DATA_BLOCK "DB_default_HMI"
{ DB_Accessible_From_Webserver := 'FALSE' ;
 S7_Optimized_Access := 'FALSE' }
VERSION : 0.1
NON_RETAIN
   STRUCT
      tALM { ExternalWritable := 'False'} : Struct   // HMI Alarms
         tE { ExternalWritable := 'False'} : Struct   // Stopping faults
            xSpare_0 { ExternalWritable := 'False'} : Bool;
            xSpare_1 { ExternalWritable := 'False'} : Bool;
            xSpare_2 { ExternalWritable := 'False'} : Bool;
            xSpare_3 { ExternalWritable := 'False'} : Bool;
            xSpare_4 { ExternalWritable := 'False'} : Bool;
            xSpare_5 { ExternalWritable := 'False'} : Bool;
            xSpare_6 { ExternalWritable := 'False'} : Bool;
            xSpare_7 { ExternalWritable := 'False'} : Bool;
            xSpare_8 { ExternalWritable := 'False'} : Bool;
            xSpare_9 { ExternalWritable := 'False'} : Bool;
            xSpare_10 { ExternalWritable := 'False'} : Bool;
            xSpare_11 { ExternalWritable := 'False'} : Bool;
            xSpare_12 { ExternalWritable := 'False'} : Bool;
            xSpare_13 { ExternalWritable := 'False'} : Bool;
            xSpare_14 { ExternalWritable := 'False'} : Bool;
            xSpare_15 { ExternalWritable := 'False'} : Bool;
            xSpare_16 { ExternalWritable := 'False'} : Bool;
            xSpare_17 { ExternalWritable := 'False'} : Bool;
            xSpare_18 { ExternalWritable := 'False'} : Bool;
            xSpare_19 { ExternalWritable := 'False'} : Bool;
            xSpare_20 { ExternalWritable := 'False'} : Bool;
            xSpare_21 { ExternalWritable := 'False'} : Bool;
            xSpare_22 { ExternalWritable := 'False'} : Bool;
            xSpare_23 { ExternalWritable := 'False'} : Bool;
            xSpare_24 { ExternalWritable := 'False'} : Bool;
            xSpare_25 { ExternalWritable := 'False'} : Bool;
            xSpare_26 { ExternalWritable := 'False'} : Bool;
            xSpare_27 { ExternalWritable := 'False'} : Bool;
            xSpare_28 { ExternalWritable := 'False'} : Bool;
            xSpare_29 { ExternalWritable := 'False'} : Bool;
            xSpare_30 { ExternalWritable := 'False'} : Bool;
            xSpare_31 { ExternalWritable := 'False'} : Bool;
         END_STRUCT;
         tS { ExternalWritable := 'False'} : Struct   // Stopping faults
            xLocalSafetySwitch { ExternalWritable := 'False'} : Bool;   // Local Safety Switch
            xFeedbackError { ExternalWritable := 'False'} : Bool;   // A171Az1.Feedback Error
            xDriveError { ExternalWritable := 'False'} : Bool;   // A171Az1.Drive Error
            xMotorFanProtection { ExternalWritable := 'False'} : Bool;   // A171QM1.Motor Fan protection
            xMotorThermalProbe { ExternalWritable := 'False'} : Bool;   // A547BT1.Motor Thermal Probe
            xSpare_5 { ExternalAccessible := 'False'; ExternalVisible := 'False'; ExternalWritable := 'False'} : Bool;
            xSpare_6 { ExternalAccessible := 'False'; ExternalVisible := 'False'; ExternalWritable := 'False'} : Bool;
            xSpare_7 { ExternalAccessible := 'False'; ExternalVisible := 'False'; ExternalWritable := 'False'} : Bool;
            xSpare_8 { ExternalAccessible := 'False'; ExternalVisible := 'False'; ExternalWritable := 'False'} : Bool;
            xSpare_9 { ExternalAccessible := 'False'; ExternalVisible := 'False'; ExternalWritable := 'False'} : Bool;
            xSpare_10 { ExternalAccessible := 'False'; ExternalVisible := 'False'; ExternalWritable := 'False'} : Bool;
            xSpare_11 { ExternalAccessible := 'False'; ExternalVisible := 'False'; ExternalWritable := 'False'} : Bool;
            xSpare_12 { ExternalAccessible := 'False'; ExternalVisible := 'False'; ExternalWritable := 'False'} : Bool;
            xSpare_13 { ExternalAccessible := 'False'; ExternalVisible := 'False'; ExternalWritable := 'False'} : Bool;
            xSpare_14 { ExternalAccessible := 'False'; ExternalVisible := 'False'; ExternalWritable := 'False'} : Bool;
            xSpare_15 { ExternalAccessible := 'False'; ExternalVisible := 'False'; ExternalWritable := 'False'} : Bool;
            xSpare_16 { ExternalAccessible := 'False'; ExternalVisible := 'False'; ExternalWritable := 'False'} : Bool;
            xSpare_17 { ExternalAccessible := 'False'; ExternalVisible := 'False'; ExternalWritable := 'False'} : Bool;
            xSpare_18 { ExternalAccessible := 'False'; ExternalVisible := 'False'; ExternalWritable := 'False'} : Bool;
            xSpare_19 { ExternalAccessible := 'False'; ExternalVisible := 'False'; ExternalWritable := 'False'} : Bool;
            xSpare_20 { ExternalAccessible := 'False'; ExternalVisible := 'False'; ExternalWritable := 'False'} : Bool;
            xSpare_21 { ExternalAccessible := 'False'; ExternalVisible := 'False'; ExternalWritable := 'False'} : Bool;
            xSpare_22 { ExternalAccessible := 'False'; ExternalVisible := 'False'; ExternalWritable := 'False'} : Bool;
            xSpare_23 { ExternalAccessible := 'False'; ExternalVisible := 'False'; ExternalWritable := 'False'} : Bool;
            xSpare_24 { ExternalAccessible := 'False'; ExternalVisible := 'False'; ExternalWritable := 'False'} : Bool;
            xSpare_25 { ExternalAccessible := 'False'; ExternalVisible := 'False'; ExternalWritable := 'False'} : Bool;
            xSpare_26 { ExternalAccessible := 'False'; ExternalVisible := 'False'; ExternalWritable := 'False'} : Bool;
            xSpare_27 { ExternalAccessible := 'False'; ExternalVisible := 'False'; ExternalWritable := 'False'} : Bool;
            xSpare_28 { ExternalAccessible := 'False'; ExternalVisible := 'False'; ExternalWritable := 'False'} : Bool;
            xSpare_29 { ExternalAccessible := 'False'; ExternalVisible := 'False'; ExternalWritable := 'False'} : Bool;
            xSpare_30 { ExternalAccessible := 'False'; ExternalVisible := 'False'; ExternalWritable := 'False'} : Bool;
            xSpare_31 { ExternalAccessible := 'False'; ExternalVisible := 'False'; ExternalWritable := 'False'} : Bool;
         END_STRUCT;
         tF { ExternalAccessible := 'False'; ExternalVisible := 'False'; ExternalWritable := 'False'} : Struct   // Faults
            xSpare_0 { ExternalAccessible := 'False'; ExternalVisible := 'False'; ExternalWritable := 'False'} : Bool;
            xSpare_1 { ExternalAccessible := 'False'; ExternalVisible := 'False'; ExternalWritable := 'False'} : Bool;
            xSpare_2 { ExternalAccessible := 'False'; ExternalVisible := 'False'; ExternalWritable := 'False'} : Bool;
            xSpare_3 { ExternalAccessible := 'False'; ExternalVisible := 'False'; ExternalWritable := 'False'} : Bool;
            xSpare_4 { ExternalAccessible := 'False'; ExternalVisible := 'False'; ExternalWritable := 'False'} : Bool;
            xSpare_5 { ExternalAccessible := 'False'; ExternalVisible := 'False'; ExternalWritable := 'False'} : Bool;
            xSpare_6 { ExternalAccessible := 'False'; ExternalVisible := 'False'; ExternalWritable := 'False'} : Bool;
            xSpare_7 { ExternalAccessible := 'False'; ExternalVisible := 'False'; ExternalWritable := 'False'} : Bool;
            xSpare_8 { ExternalAccessible := 'False'; ExternalVisible := 'False'; ExternalWritable := 'False'} : Bool;
            xSpare_9 { ExternalAccessible := 'False'; ExternalVisible := 'False'; ExternalWritable := 'False'} : Bool;
            xSpare_10 { ExternalAccessible := 'False'; ExternalVisible := 'False'; ExternalWritable := 'False'} : Bool;
            xSpare_11 { ExternalAccessible := 'False'; ExternalVisible := 'False'; ExternalWritable := 'False'} : Bool;
            xSpare_12 { ExternalAccessible := 'False'; ExternalVisible := 'False'; ExternalWritable := 'False'} : Bool;
            xSpare_13 { ExternalAccessible := 'False'; ExternalVisible := 'False'; ExternalWritable := 'False'} : Bool;
            xSpare_14 { ExternalAccessible := 'False'; ExternalVisible := 'False'; ExternalWritable := 'False'} : Bool;
            xSpare_15 { ExternalAccessible := 'False'; ExternalVisible := 'False'; ExternalWritable := 'False'} : Bool;
            xSpare_16 { ExternalAccessible := 'False'; ExternalVisible := 'False'; ExternalWritable := 'False'} : Bool;
            xSpare_17 { ExternalAccessible := 'False'; ExternalVisible := 'False'; ExternalWritable := 'False'} : Bool;
            xSpare_18 { ExternalAccessible := 'False'; ExternalVisible := 'False'; ExternalWritable := 'False'} : Bool;
            xSpare_19 { ExternalAccessible := 'False'; ExternalVisible := 'False'; ExternalWritable := 'False'} : Bool;
            xSpare_20 { ExternalAccessible := 'False'; ExternalVisible := 'False'; ExternalWritable := 'False'} : Bool;
            xSpare_21 { ExternalAccessible := 'False'; ExternalVisible := 'False'; ExternalWritable := 'False'} : Bool;
            xSpare_22 { ExternalAccessible := 'False'; ExternalVisible := 'False'; ExternalWritable := 'False'} : Bool;
            xSpare_23 { ExternalAccessible := 'False'; ExternalVisible := 'False'; ExternalWritable := 'False'} : Bool;
            xSpare_24 { ExternalAccessible := 'False'; ExternalVisible := 'False'; ExternalWritable := 'False'} : Bool;
            xSpare_25 { ExternalAccessible := 'False'; ExternalVisible := 'False'; ExternalWritable := 'False'} : Bool;
            xSpare_26 { ExternalAccessible := 'False'; ExternalVisible := 'False'; ExternalWritable := 'False'} : Bool;
            xSpare_27 { ExternalAccessible := 'False'; ExternalVisible := 'False'; ExternalWritable := 'False'} : Bool;
            xSpare_28 { ExternalAccessible := 'False'; ExternalVisible := 'False'; ExternalWritable := 'False'} : Bool;
            xSpare_29 { ExternalAccessible := 'False'; ExternalVisible := 'False'; ExternalWritable := 'False'} : Bool;
            xSpare_30 { ExternalAccessible := 'False'; ExternalVisible := 'False'; ExternalWritable := 'False'} : Bool;
            xSpare_31 { ExternalAccessible := 'False'; ExternalVisible := 'False'; ExternalWritable := 'False'} : Bool;
         END_STRUCT;
         tW { ExternalAccessible := 'False'; ExternalVisible := 'False'; ExternalWritable := 'False'} : Struct   // Warnings
            xSpare_0 { ExternalAccessible := 'False'; ExternalVisible := 'False'; ExternalWritable := 'False'} : Bool;
            xSpare_1 { ExternalAccessible := 'False'; ExternalVisible := 'False'; ExternalWritable := 'False'} : Bool;
            xSpare_2 { ExternalAccessible := 'False'; ExternalVisible := 'False'; ExternalWritable := 'False'} : Bool;
            xSpare_3 { ExternalAccessible := 'False'; ExternalVisible := 'False'; ExternalWritable := 'False'} : Bool;
            xSpare_4 { ExternalAccessible := 'False'; ExternalVisible := 'False'; ExternalWritable := 'False'} : Bool;
            xSpare_5 { ExternalAccessible := 'False'; ExternalVisible := 'False'; ExternalWritable := 'False'} : Bool;
            xSpare_6 { ExternalAccessible := 'False'; ExternalVisible := 'False'; ExternalWritable := 'False'} : Bool;
            xSpare_7 { ExternalAccessible := 'False'; ExternalVisible := 'False'; ExternalWritable := 'False'} : Bool;
            xSpare_8 { ExternalAccessible := 'False'; ExternalVisible := 'False'; ExternalWritable := 'False'} : Bool;
            xSpare_9 { ExternalAccessible := 'False'; ExternalVisible := 'False'; ExternalWritable := 'False'} : Bool;
            xSpare_10 { ExternalAccessible := 'False'; ExternalVisible := 'False'; ExternalWritable := 'False'} : Bool;
            xSpare_11 { ExternalAccessible := 'False'; ExternalVisible := 'False'; ExternalWritable := 'False'} : Bool;
            xSpare_12 { ExternalAccessible := 'False'; ExternalVisible := 'False'; ExternalWritable := 'False'} : Bool;
            xSpare_13 { ExternalAccessible := 'False'; ExternalVisible := 'False'; ExternalWritable := 'False'} : Bool;
            xSpare_14 { ExternalAccessible := 'False'; ExternalVisible := 'False'; ExternalWritable := 'False'} : Bool;
            xSpare_15 { ExternalAccessible := 'False'; ExternalVisible := 'False'; ExternalWritable := 'False'} : Bool;
            xSpare_16 { ExternalAccessible := 'False'; ExternalVisible := 'False'; ExternalWritable := 'False'} : Bool;
            xSpare_17 { ExternalAccessible := 'False'; ExternalVisible := 'False'; ExternalWritable := 'False'} : Bool;
            xSpare_18 { ExternalAccessible := 'False'; ExternalVisible := 'False'; ExternalWritable := 'False'} : Bool;
            xSpare_19 { ExternalAccessible := 'False'; ExternalVisible := 'False'; ExternalWritable := 'False'} : Bool;
            xSpare_20 { ExternalAccessible := 'False'; ExternalVisible := 'False'; ExternalWritable := 'False'} : Bool;
            xSpare_21 { ExternalAccessible := 'False'; ExternalVisible := 'False'; ExternalWritable := 'False'} : Bool;
            xSpare_22 { ExternalAccessible := 'False'; ExternalVisible := 'False'; ExternalWritable := 'False'} : Bool;
            xSpare_23 { ExternalAccessible := 'False'; ExternalVisible := 'False'; ExternalWritable := 'False'} : Bool;
            xSpare_24 { ExternalAccessible := 'False'; ExternalVisible := 'False'; ExternalWritable := 'False'} : Bool;
            xSpare_25 { ExternalAccessible := 'False'; ExternalVisible := 'False'; ExternalWritable := 'False'} : Bool;
            xSpare_26 { ExternalAccessible := 'False'; ExternalVisible := 'False'; ExternalWritable := 'False'} : Bool;
            xSpare_27 { ExternalAccessible := 'False'; ExternalVisible := 'False'; ExternalWritable := 'False'} : Bool;
            xSpare_28 { ExternalAccessible := 'False'; ExternalVisible := 'False'; ExternalWritable := 'False'} : Bool;
            xSpare_29 { ExternalAccessible := 'False'; ExternalVisible := 'False'; ExternalWritable := 'False'} : Bool;
            xSpare_30 { ExternalAccessible := 'False'; ExternalVisible := 'False'; ExternalWritable := 'False'} : Bool;
            xSpare_31 { ExternalAccessible := 'False'; ExternalVisible := 'False'; ExternalWritable := 'False'} : Bool;
         END_STRUCT;
      END_STRUCT;
      tHMR { ExternalWritable := 'False'} : Struct   // HMI Read
         xSpare0 { ExternalWritable := 'False'} : Bool;
         xSpare1 { ExternalWritable := 'False'} : Bool;
         xSpare2 { ExternalWritable := 'False'} : Bool;
         xSpare3 { ExternalWritable := 'False'} : Bool;
         xSpare4 { ExternalWritable := 'False'} : Bool;
         xSpare5 { ExternalWritable := 'False'} : Bool;
         xSpare6 { ExternalWritable := 'False'} : Bool;
         xSpare7 { ExternalWritable := 'False'} : Bool;
         xSpare8 { ExternalWritable := 'False'} : Bool;
         xSpare9 { ExternalWritable := 'False'} : Bool;
         xSpare10 { ExternalWritable := 'False'} : Bool;
         xSpare11 { ExternalWritable := 'False'} : Bool;
         xSpare12 { ExternalWritable := 'False'} : Bool;
         xSpare13 { ExternalWritable := 'False'} : Bool;
         xManualCommandEnabled { ExternalWritable := 'False'} : Bool;   // Manual Command enabled {x|x|x|x|O}
         xSpare15 { ExternalWritable := 'False'} : Bool;
         xSpare16 { ExternalWritable := 'False'} : Bool;
         xSpare17 { ExternalWritable := 'False'} : Bool;
         xSpare18 { ExternalWritable := 'False'} : Bool;
         xSpare19 { ExternalWritable := 'False'} : Bool;
         xSpare20 { ExternalWritable := 'False'} : Bool;
         xSpare21 { ExternalWritable := 'False'} : Bool;
         xSpare22 { ExternalWritable := 'False'} : Bool;
         xSpare23 { ExternalWritable := 'False'} : Bool;
         xSpare24 { ExternalWritable := 'False'} : Bool;
         xSpare25 { ExternalWritable := 'False'} : Bool;
         xSpare26 { ExternalWritable := 'False'} : Bool;
         xSpare27 { ExternalWritable := 'False'} : Bool;
         xSpare28 { ExternalWritable := 'False'} : Bool;
         xSpare29 { ExternalWritable := 'False'} : Bool;
         xSpare30 { ExternalWritable := 'False'} : Bool;
         xSpare31 { ExternalWritable := 'False'} : Bool;
         xSpare { ExternalWritable := 'False'} : Array[0..15] of Bool;
         iSpare0 { ExternalWritable := 'False'} : Int;
         iSpare1 { ExternalWritable := 'False'} : Int;
         iSpare2 { ExternalWritable := 'False'} : Int;
         iSpare3 { ExternalWritable := 'False'} : Int;
         iSpare4 { ExternalWritable := 'False'} : Int;
         iSpare5 { ExternalWritable := 'False'} : Int;
         iSpare6 { ExternalWritable := 'False'} : Int;
         iSpare7 { ExternalWritable := 'False'} : Int;
         iSpare8 { ExternalWritable := 'False'} : Int;
         iSpare9 { ExternalWritable := 'False'} : Int;
         iSpare10 { ExternalWritable := 'False'} : Int;
         iSpare11 { ExternalWritable := 'False'} : Int;
         iSpare12 { ExternalWritable := 'False'} : Int;
         iSpare13 { ExternalWritable := 'False'} : Int;
         iSpare14 { ExternalWritable := 'False'} : Int;
         iSpare15 { ExternalWritable := 'False'} : Int;
         iSpare16 { ExternalWritable := 'False'} : Int;
         dSpare0 { ExternalWritable := 'False'} : DInt;   //
         dSpare1 { ExternalWritable := 'False'} : DInt;   //
         dSpare2 { ExternalWritable := 'False'} : DInt;
         dSpare3 { ExternalWritable := 'False'} : DInt;
         dSpare4 { ExternalWritable := 'False'} : DInt;
         dSpare5 { ExternalWritable := 'False'} : DInt;
         dSpare6 { ExternalWritable := 'False'} : DInt;
         dSpare7 { ExternalWritable := 'False'} : DInt;
         dSpare8 { ExternalWritable := 'False'} : DInt;
         dSpare9 { ExternalWritable := 'False'} : DInt;
         dSpare10 { ExternalWritable := 'False'} : DInt;
         dSpare11 { ExternalWritable := 'False'} : DInt;
         dSpare12 { ExternalWritable := 'False'} : DInt;
         dSpare13 { ExternalWritable := 'False'} : DInt;
         dSpare14 { ExternalWritable := 'False'} : DInt;
         dSpare15 { ExternalWritable := 'False'} : DInt;
         rSpare0 { ExternalWritable := 'False'} : Real;
         rSpare1 { ExternalWritable := 'False'} : Real;
         rSpare2 { ExternalWritable := 'False'} : Real;
         rSpare3 { ExternalWritable := 'False'} : Real;
         rSpare4 { ExternalWritable := 'False'} : Real;
         rSpare5 { ExternalWritable := 'False'} : Real;
         rSpare6 { ExternalWritable := 'False'} : Real;
         rSpare7 { ExternalWritable := 'False'} : Real;
         rSpare8 { ExternalWritable := 'False'} : Real;
         tManCmd { ExternalWritable := 'False'} : Struct
            xSpare0 { ExternalWritable := 'False'} : Bool;   //
            xSpare1 { ExternalWritable := 'False'} : Bool;
            xSpare2 { ExternalWritable := 'False'} : Bool;
            xSpare3 { ExternalWritable := 'False'} : Bool;
            xSpare4 { ExternalWritable := 'False'} : Bool;
            xSpare5 { ExternalWritable := 'False'} : Bool;
            xSpare6 { ExternalWritable := 'False'} : Bool;
            xSpare7 { ExternalWritable := 'False'} : Bool;
            xSpare8 { ExternalWritable := 'False'} : Bool;
            xSpare9 { ExternalWritable := 'False'} : Bool;
            xSpare10 { ExternalWritable := 'False'} : Bool;
            xSpare11 { ExternalWritable := 'False'} : Bool;
            xSpare12 { ExternalWritable := 'False'} : Bool;
            xSpare13 { ExternalWritable := 'False'} : Bool;
            xSpare14 { ExternalWritable := 'False'} : Bool;
            xSpare15 { ExternalWritable := 'False'} : Bool;
            xSpare { ExternalWritable := 'False'} : Array[0..15] of Bool;
         END_STRUCT;
      END_STRUCT;
      tHMW : Struct   // HMI Write
         xSpare0 : Bool;   //
         xSpare1 : Bool;
         xSpare2 : Bool;
         xSpare3 : Bool;
         xSpare4 : Bool;
         xSpare5 : Bool;
         xSpare6 : Bool;
         xSpare7 : Bool;
         xSpare8 : Bool;
         xSpare9 : Bool;
         xSpare10 : Bool;   //
         xSpare11 : Bool;
         xSpare12 : Bool;
         xSpare13 : Bool;
         xEnableManualCommand : Bool;   // Enable Disable Manual command {x|x|x|x|O}
         xSpare15 : Bool;
         xSpare16 : Bool;
         xSpare17 : Bool;
         xSpare18 : Bool;
         xSpare19 : Bool;
         xSpare20 : Bool;
         xSpare21 : Bool;
         xSpare22 : Bool;
         xSpare23 : Bool;
         xSpare24 : Bool;
         xSpare25 : Bool;
         xSpare26 : Bool;
         xSpare27 : Bool;
         xSpare28 : Bool;
         xSpare29 : Bool;
         xSpare30 : Bool;
         xSpare31 : Bool;
         xSpare : Array[0..15] of Bool;
         iSpare0 : Int;
         iSpare1 : Int;
         iSpare2 : Int;
         iSpare3 : Int;
         iSpare4 : Int;
         iSpare5 : Int;
         iSpare6 : Int;
         iSpare7 : Int;
         iSpare8 : Int;
         iSpare9 : Int;
         iSpare10 : Int;
         iSpare11 : Int;
         iSpare12 : Int;
         iSpare13 : Int;
         iSpare14 : Int;
         iSpare15 : Int;
         iSpare16 : Int;
         dSpare0 : DInt;   //
         dSpare1 : DInt;   //
         dSpare2 : DInt;   //
         dSpare3 : DInt;
         dSpare4 : DInt;
         dSpare5 : DInt;
         dSpare6 : DInt;
         dSpare7 : DInt;
         dSpare8 : DInt;
         dSpare9 : DInt;
         dSpare10 : DInt;
         dSpare11 : DInt;
         dSpare12 : DInt;
         dSpare13 : DInt;
         dSpare14 : DInt;
         dSpare15 : DInt;
         dSpare16 : DInt;
         rSpare0 : Real;
         rSpare1 : Real;
         rSpare2 : Real;
         rSpare3 : Real;
         rSpare4 : Real;
         rSpare5 : Real;
         rSpare6 : Real;
         rSpare7 : Real;
         rSpare8 : Real;
         tManCmd : Struct
            xSpare0 : Bool;   //
            xSpare1 : Bool;
            xSpare2 { ExternalWritable := 'False'} : Bool;
            xSpare3 { ExternalWritable := 'False'} : Bool;
            xSpare4 { ExternalWritable := 'False'} : Bool;
            xSpare5 { ExternalWritable := 'False'} : Bool;
            xSpare6 { ExternalWritable := 'False'} : Bool;
            xSpare7 { ExternalWritable := 'False'} : Bool;
            xSpare8 { ExternalWritable := 'False'} : Bool;
            xSpare9 { ExternalWritable := 'False'} : Bool;
            xSpare10 { ExternalWritable := 'False'} : Bool;
            xSpare11 { ExternalWritable := 'False'} : Bool;
            xSpare12 { ExternalWritable := 'False'} : Bool;
            xSpare13 { ExternalWritable := 'False'} : Bool;
            xSpare14 { ExternalWritable := 'False'} : Bool;
            xSpare15 { ExternalWritable := 'False'} : Bool;
            xSpare16 : Bool;
            xSpare17 : Bool;
            xSpare18 : Bool;
            xSpare19 : Bool;
            xSpare20 : Bool;
            xSpare21 : Bool;
            xSpare22 : Bool;
            xSpare23 : Bool;
            xSpare24 : Bool;
            xSpare25 : Bool;
            xSpare26 : Bool;
            xSpare27 : Bool;
            xSpare28 : Bool;
            xSpare29 : Bool;
            xSpare30 : Bool;
            xSpare31 : Bool;
         END_STRUCT;
      END_STRUCT;
   END_STRUCT;


BEGIN

END_DATA_BLOCK

DATA_BLOCK "DB_M220_3_HMI"
{ DB_Accessible_From_Webserver := 'FALSE' ;
 S7_Optimized_Access := 'FALSE' }
VERSION : 0.1
NON_RETAIN
   STRUCT
      tALM { ExternalWritable := 'False'} : Struct   // HMI Alarms
         tE { ExternalWritable := 'False'} : Struct   // Stopping faults
            xSpare_0 { ExternalWritable := 'False'} : Bool;
            xSpare_1 { ExternalWritable := 'False'} : Bool;
            xSpare_2 { ExternalWritable := 'False'} : Bool;
            xSpare_3 { ExternalWritable := 'False'} : Bool;
            xSpare_4 { ExternalWritable := 'False'} : Bool;
            xSpare_5 { ExternalWritable := 'False'} : Bool;
            xSpare_6 { ExternalWritable := 'False'} : Bool;
            xSpare_7 { ExternalWritable := 'False'} : Bool;
            xSpare_8 { ExternalWritable := 'False'} : Bool;
            xSpare_9 { ExternalWritable := 'False'} : Bool;
            xSpare_10 { ExternalWritable := 'False'} : Bool;
            xSpare_11 { ExternalWritable := 'False'} : Bool;
            xSpare_12 { ExternalWritable := 'False'} : Bool;
            xSpare_13 { ExternalWritable := 'False'} : Bool;
            xSpare_14 { ExternalWritable := 'False'} : Bool;
            xSpare_15 { ExternalWritable := 'False'} : Bool;
            xSpare_16 { ExternalWritable := 'False'} : Bool;
            xSpare_17 { ExternalWritable := 'False'} : Bool;
            xSpare_18 { ExternalWritable := 'False'} : Bool;
            xSpare_19 { ExternalWritable := 'False'} : Bool;
            xSpare_20 { ExternalWritable := 'False'} : Bool;
            xSpare_21 { ExternalWritable := 'False'} : Bool;
            xSpare_22 { ExternalWritable := 'False'} : Bool;
            xSpare_23 { ExternalWritable := 'False'} : Bool;
            xSpare_24 { ExternalWritable := 'False'} : Bool;
            xSpare_25 { ExternalWritable := 'False'} : Bool;
            xSpare_26 { ExternalWritable := 'False'} : Bool;
            xSpare_27 { ExternalWritable := 'False'} : Bool;
            xSpare_28 { ExternalWritable := 'False'} : Bool;
            xSpare_29 { ExternalWritable := 'False'} : Bool;
            xSpare_30 { ExternalWritable := 'False'} : Bool;
            xSpare_31 { ExternalWritable := 'False'} : Bool;
         END_STRUCT;
         tS { ExternalWritable := 'False'} : Struct
            x0 { ExternalWritable := 'False'} : Bool;   // AZ.Carriage homing timeout
            x1 { ExternalWritable := 'False'} : Bool;   // AZ.Carriage positioning timeout
            x2 { ExternalWritable := 'False'} : Bool;   // QM.Carriage translation overload cutout
            x3 { ExternalWritable := 'False'} : Bool;   // SQ.Forward overstroke translation
            x4 { ExternalWritable := 'False'} : Bool;   // SQ.Backward overstroke translation
            x5 { ExternalWritable := 'False'} : Bool;   // AZ.Feedback error
            x6 { ExternalWritable := 'False'} : Bool;   // AZ.Drive not enable
            x7 { ExternalWritable := 'False'} : Bool;   // AZ.Drive not ok
            x8 { ExternalWritable := 'False'} : Bool;   // AZ.Drive link timeout
            x9 { ExternalWritable := 'False'} : Bool;
            x10 { ExternalWritable := 'False'} : Bool;
            x11 { ExternalWritable := 'False'} : Bool;
            x12 { ExternalWritable := 'False'} : Bool;
            x13 { ExternalWritable := 'False'} : Bool;
            x14 { ExternalWritable := 'False'} : Bool;
            x15 { ExternalWritable := 'False'} : Bool;
            x16 { ExternalWritable := 'False'} : Bool;
            x17 { ExternalWritable := 'False'} : Bool;
            x18 { ExternalWritable := 'False'} : Bool;
            x19 { ExternalWritable := 'False'} : Bool;
            x20 { ExternalWritable := 'False'} : Bool;
            x21 { ExternalWritable := 'False'} : Bool;
            x22 { ExternalWritable := 'False'} : Bool;
            x23 { ExternalWritable := 'False'} : Bool;
            x24 { ExternalWritable := 'False'} : Bool;
            x25 { ExternalWritable := 'False'} : Bool;
            x26 { ExternalWritable := 'False'} : Bool;
            x27 { ExternalWritable := 'False'} : Bool;
            x28 { ExternalWritable := 'False'} : Bool;
            x29 { ExternalWritable := 'False'} : Bool;
            x30 { ExternalWritable := 'False'} : Bool;
            x31 { ExternalWritable := 'False'} : Bool;
         END_STRUCT;
         tF { ExternalAccessible := 'False'; ExternalVisible := 'False'; ExternalWritable := 'False'} : Struct   // Faults
            xSpare_0 { ExternalAccessible := 'False'; ExternalVisible := 'False'; ExternalWritable := 'False'} : Bool;
            xSpare_1 { ExternalAccessible := 'False'; ExternalVisible := 'False'; ExternalWritable := 'False'} : Bool;
            xSpare_2 { ExternalAccessible := 'False'; ExternalVisible := 'False'; ExternalWritable := 'False'} : Bool;
            xSpare_3 { ExternalAccessible := 'False'; ExternalVisible := 'False'; ExternalWritable := 'False'} : Bool;
            xSpare_4 { ExternalAccessible := 'False'; ExternalVisible := 'False'; ExternalWritable := 'False'} : Bool;
            xSpare_5 { ExternalAccessible := 'False'; ExternalVisible := 'False'; ExternalWritable := 'False'} : Bool;
            xSpare_6 { ExternalAccessible := 'False'; ExternalVisible := 'False'; ExternalWritable := 'False'} : Bool;
            xSpare_7 { ExternalAccessible := 'False'; ExternalVisible := 'False'; ExternalWritable := 'False'} : Bool;
            xSpare_8 { ExternalAccessible := 'False'; ExternalVisible := 'False'; ExternalWritable := 'False'} : Bool;
            xSpare_9 { ExternalAccessible := 'False'; ExternalVisible := 'False'; ExternalWritable := 'False'} : Bool;
            xSpare_10 { ExternalAccessible := 'False'; ExternalVisible := 'False'; ExternalWritable := 'False'} : Bool;
            xSpare_11 { ExternalAccessible := 'False'; ExternalVisible := 'False'; ExternalWritable := 'False'} : Bool;
            xSpare_12 { ExternalAccessible := 'False'; ExternalVisible := 'False'; ExternalWritable := 'False'} : Bool;
            xSpare_13 { ExternalAccessible := 'False'; ExternalVisible := 'False'; ExternalWritable := 'False'} : Bool;
            xSpare_14 { ExternalAccessible := 'False'; ExternalVisible := 'False'; ExternalWritable := 'False'} : Bool;
            xSpare_15 { ExternalAccessible := 'False'; ExternalVisible := 'False'; ExternalWritable := 'False'} : Bool;
            xSpare_16 { ExternalAccessible := 'False'; ExternalVisible := 'False'; ExternalWritable := 'False'} : Bool;
            xSpare_17 { ExternalAccessible := 'False'; ExternalVisible := 'False'; ExternalWritable := 'False'} : Bool;
            xSpare_18 { ExternalAccessible := 'False'; ExternalVisible := 'False'; ExternalWritable := 'False'} : Bool;
            xSpare_19 { ExternalAccessible := 'False'; ExternalVisible := 'False'; ExternalWritable := 'False'} : Bool;
            xSpare_20 { ExternalAccessible := 'False'; ExternalVisible := 'False'; ExternalWritable := 'False'} : Bool;
            xSpare_21 { ExternalAccessible := 'False'; ExternalVisible := 'False'; ExternalWritable := 'False'} : Bool;
            xSpare_22 { ExternalAccessible := 'False'; ExternalVisible := 'False'; ExternalWritable := 'False'} : Bool;
            xSpare_23 { ExternalAccessible := 'False'; ExternalVisible := 'False'; ExternalWritable := 'False'} : Bool;
            xSpare_24 { ExternalAccessible := 'False'; ExternalVisible := 'False'; ExternalWritable := 'False'} : Bool;
            xSpare_25 { ExternalAccessible := 'False'; ExternalVisible := 'False'; ExternalWritable := 'False'} : Bool;
            xSpare_26 { ExternalAccessible := 'False'; ExternalVisible := 'False'; ExternalWritable := 'False'} : Bool;
            xSpare_27 { ExternalAccessible := 'False'; ExternalVisible := 'False'; ExternalWritable := 'False'} : Bool;
            xSpare_28 { ExternalAccessible := 'False'; ExternalVisible := 'False'; ExternalWritable := 'False'} : Bool;
            xSpare_29 { ExternalAccessible := 'False'; ExternalVisible := 'False'; ExternalWritable := 'False'} : Bool;
            xSpare_30 { ExternalAccessible := 'False'; ExternalVisible := 'False'; ExternalWritable := 'False'} : Bool;
            xSpare_31 { ExternalAccessible := 'False'; ExternalVisible := 'False'; ExternalWritable := 'False'} : Bool;
         END_STRUCT;
         tW { ExternalAccessible := 'False'; ExternalVisible := 'False'; ExternalWritable := 'False'} : Struct   // Warnings
            xSpare_0 { ExternalAccessible := 'False'; ExternalVisible := 'False'; ExternalWritable := 'False'} : Bool;
            xSpare_1 { ExternalAccessible := 'False'; ExternalVisible := 'False'; ExternalWritable := 'False'} : Bool;
            xSpare_2 { ExternalAccessible := 'False'; ExternalVisible := 'False'; ExternalWritable := 'False'} : Bool;
            xSpare_3 { ExternalAccessible := 'False'; ExternalVisible := 'False'; ExternalWritable := 'False'} : Bool;
            xSpare_4 { ExternalAccessible := 'False'; ExternalVisible := 'False'; ExternalWritable := 'False'} : Bool;
            xSpare_5 { ExternalAccessible := 'False'; ExternalVisible := 'False'; ExternalWritable := 'False'} : Bool;
            xSpare_6 { ExternalAccessible := 'False'; ExternalVisible := 'False'; ExternalWritable := 'False'} : Bool;
            xSpare_7 { ExternalAccessible := 'False'; ExternalVisible := 'False'; ExternalWritable := 'False'} : Bool;
            xSpare_8 { ExternalAccessible := 'False'; ExternalVisible := 'False'; ExternalWritable := 'False'} : Bool;
            xSpare_9 { ExternalAccessible := 'False'; ExternalVisible := 'False'; ExternalWritable := 'False'} : Bool;
            xSpare_10 { ExternalAccessible := 'False'; ExternalVisible := 'False'; ExternalWritable := 'False'} : Bool;
            xSpare_11 { ExternalAccessible := 'False'; ExternalVisible := 'False'; ExternalWritable := 'False'} : Bool;
            xSpare_12 { ExternalAccessible := 'False'; ExternalVisible := 'False'; ExternalWritable := 'False'} : Bool;
            xSpare_13 { ExternalAccessible := 'False'; ExternalVisible := 'False'; ExternalWritable := 'False'} : Bool;
            xSpare_14 { ExternalAccessible := 'False'; ExternalVisible := 'False'; ExternalWritable := 'False'} : Bool;
            xSpare_15 { ExternalAccessible := 'False'; ExternalVisible := 'False'; ExternalWritable := 'False'} : Bool;
            xSpare_16 { ExternalAccessible := 'False'; ExternalVisible := 'False'; ExternalWritable := 'False'} : Bool;
            xSpare_17 { ExternalAccessible := 'False'; ExternalVisible := 'False'; ExternalWritable := 'False'} : Bool;
            xSpare_18 { ExternalAccessible := 'False'; ExternalVisible := 'False'; ExternalWritable := 'False'} : Bool;
            xSpare_19 { ExternalAccessible := 'False'; ExternalVisible := 'False'; ExternalWritable := 'False'} : Bool;
            xSpare_20 { ExternalAccessible := 'False'; ExternalVisible := 'False'; ExternalWritable := 'False'} : Bool;
            xSpare_21 { ExternalAccessible := 'False'; ExternalVisible := 'False'; ExternalWritable := 'False'} : Bool;
            xSpare_22 { ExternalAccessible := 'False'; ExternalVisible := 'False'; ExternalWritable := 'False'} : Bool;
            xSpare_23 { ExternalAccessible := 'False'; ExternalVisible := 'False'; ExternalWritable := 'False'} : Bool;
            xSpare_24 { ExternalAccessible := 'False'; ExternalVisible := 'False'; ExternalWritable := 'False'} : Bool;
            xSpare_25 { ExternalAccessible := 'False'; ExternalVisible := 'False'; ExternalWritable := 'False'} : Bool;
            xSpare_26 { ExternalAccessible := 'False'; ExternalVisible := 'False'; ExternalWritable := 'False'} : Bool;
            xSpare_27 { ExternalAccessible := 'False'; ExternalVisible := 'False'; ExternalWritable := 'False'} : Bool;
            xSpare_28 { ExternalAccessible := 'False'; ExternalVisible := 'False'; ExternalWritable := 'False'} : Bool;
            xSpare_29 { ExternalAccessible := 'False'; ExternalVisible := 'False'; ExternalWritable := 'False'} : Bool;
            xSpare_30 { ExternalAccessible := 'False'; ExternalVisible := 'False'; ExternalWritable := 'False'} : Bool;
            xSpare_31 { ExternalAccessible := 'False'; ExternalVisible := 'False'; ExternalWritable := 'False'} : Bool;
         END_STRUCT;
      END_STRUCT;
      tHMR { ExternalWritable := 'False'} : Struct   // HMI Read
         xCalibrationsAllowed { ExternalWritable := 'False'} : Bool;   // Calibrations allowed {x|x|x|x|O}
         xSpare1 { ExternalWritable := 'False'} : Bool;
         xSpare2 { ExternalWritable := 'False'} : Bool;
         xSpare3 { ExternalWritable := 'False'} : Bool;
         xSpare4 { ExternalWritable := 'False'} : Bool;
         xSpare5 { ExternalWritable := 'False'} : Bool;
         xSpare6 { ExternalWritable := 'False'} : Bool;
         xSpare7 { ExternalWritable := 'False'} : Bool;
         xSpare8 { ExternalWritable := 'False'} : Bool;
         xSpare9 { ExternalWritable := 'False'} : Bool;
         xSpare10 { ExternalWritable := 'False'} : Bool;
         xSpare11 { ExternalWritable := 'False'} : Bool;
         xSpare12 { ExternalWritable := 'False'} : Bool;
         xSpare13 { ExternalWritable := 'False'} : Bool;
         xSpare14 { ExternalWritable := 'False'} : Bool;   //
         xSpare15 { ExternalWritable := 'False'} : Bool;
         xSpare16 { ExternalWritable := 'False'} : Bool;
         xSpare17 { ExternalWritable := 'False'} : Bool;
         xSpare18 { ExternalWritable := 'False'} : Bool;
         xSpare19 { ExternalWritable := 'False'} : Bool;
         xSpare20 { ExternalWritable := 'False'} : Bool;
         xSpare21 { ExternalWritable := 'False'} : Bool;
         xSpare22 { ExternalWritable := 'False'} : Bool;
         xSpare23 { ExternalWritable := 'False'} : Bool;
         xSpare24 { ExternalWritable := 'False'} : Bool;
         xSpare25 { ExternalWritable := 'False'} : Bool;
         xSpare26 { ExternalWritable := 'False'} : Bool;
         xSpare27 { ExternalWritable := 'False'} : Bool;
         xSpare28 { ExternalWritable := 'False'} : Bool;
         xSpare29 { ExternalWritable := 'False'} : Bool;
         xSpare30 { ExternalWritable := 'False'} : Bool;
         xSpare31 { ExternalWritable := 'False'} : Bool;
         xSpare { ExternalWritable := 'False'} : Array[0..15] of Bool;
         iSpare0 { ExternalWritable := 'False'} : Int;
         iSpare1 { ExternalWritable := 'False'} : Int;
         iSpare2 { ExternalWritable := 'False'} : Int;
         iSpare3 { ExternalWritable := 'False'} : Int;
         iSpare4 { ExternalWritable := 'False'} : Int;
         iSpare5 { ExternalWritable := 'False'} : Int;
         iSpare6 { ExternalWritable := 'False'} : Int;
         iSpare7 { ExternalWritable := 'False'} : Int;
         iSpare8 { ExternalWritable := 'False'} : Int;
         iSpare9 { ExternalWritable := 'False'} : Int;
         iSpare10 { ExternalWritable := 'False'} : Int;
         iSpare11 { ExternalWritable := 'False'} : Int;
         iSpare12 { ExternalWritable := 'False'} : Int;
         iSpare13 { ExternalWritable := 'False'} : Int;
         iSpare14 { ExternalWritable := 'False'} : Int;
         iSpare15 { ExternalWritable := 'False'} : Int;
         iSpare16 { ExternalWritable := 'False'} : Int;
         dCarriageStatus { ExternalWritable := 'False'} : DInt;   // Carriage status (1=Not Initialized 2=Not referred 3=Not positioned 4=Positioned 5=Positioning 6=Virtual collision 7=Anomaly) {x|x|x|x|O}
         dCarriageHomePosition_cmm { ExternalWritable := 'False'} : DInt;   // Carriage home position [mm/100] {mm/100|mm|x|x|O}
         dCarriageActualPosition_cmm { ExternalWritable := 'False'} : DInt;   // Carriage actual position [mm/100] {mm/100|mm|x|x|O}
         dSpare3 { ExternalWritable := 'False'} : DInt;
         dSpare4 { ExternalWritable := 'False'} : DInt;
         dSpare5 { ExternalWritable := 'False'} : DInt;
         dSpare6 { ExternalWritable := 'False'} : DInt;
         dSpare7 { ExternalWritable := 'False'} : DInt;
         dSpare8 { ExternalWritable := 'False'} : DInt;
         dSpare9 { ExternalWritable := 'False'} : DInt;
         dSpare10 { ExternalWritable := 'False'} : DInt;
         dSpare11 { ExternalWritable := 'False'} : DInt;
         dSpare12 { ExternalWritable := 'False'} : DInt;
         dSpare13 { ExternalWritable := 'False'} : DInt;
         dSpare14 { ExternalWritable := 'False'} : DInt;
         dSpare15 { ExternalWritable := 'False'} : DInt;
         rSpare0 { ExternalWritable := 'False'} : Real;
         rSpare1 { ExternalWritable := 'False'} : Real;
         rSpare2 { ExternalWritable := 'False'} : Real;
         rSpare3 { ExternalWritable := 'False'} : Real;
         rSpare4 { ExternalWritable := 'False'} : Real;
         rSpare5 { ExternalWritable := 'False'} : Real;
         rSpare6 { ExternalWritable := 'False'} : Real;
         rSpare7 { ExternalWritable := 'False'} : Real;
         rSpare8 { ExternalWritable := 'False'} : Real;
         tManCmd { ExternalWritable := 'False'} : Struct
            xJogForward { ExternalWritable := 'False'} : Bool;   // Carriage manual jog forward fdbk {x|x|x|x|O}
            xJogBackward { ExternalWritable := 'False'} : Bool;   // Carriage manual jog backward fdbk {x|x|x|x|O}
            xSpare2 { ExternalWritable := 'False'} : Bool;
            xSpare3 { ExternalWritable := 'False'} : Bool;
            xSpare4 { ExternalWritable := 'False'} : Bool;
            xSpare5 { ExternalWritable := 'False'} : Bool;
            xSpare6 { ExternalWritable := 'False'} : Bool;
            xSpare7 { ExternalWritable := 'False'} : Bool;
            xSpare8 { ExternalWritable := 'False'} : Bool;
            xSpare9 { ExternalWritable := 'False'} : Bool;
            xSpare10 { ExternalWritable := 'False'} : Bool;
            xSpare11 { ExternalWritable := 'False'} : Bool;
            xSpare12 { ExternalWritable := 'False'} : Bool;
            xSpare13 { ExternalWritable := 'False'} : Bool;
            xSpare14 { ExternalWritable := 'False'} : Bool;
            xSpare15 { ExternalWritable := 'False'} : Bool;
            xSpare { ExternalWritable := 'False'} : Array[0..15] of Bool;
         END_STRUCT;
      END_STRUCT;
      tHMW : Struct   // HMI Write
         xForceCarriageHoming : Bool;   // Force the homing of the carriage {x|x|x|x|M}
         xSpare1 : Bool;
         xSpare2 : Bool;
         xSpare3 : Bool;
         xSpare4 : Bool;
         xSpare5 : Bool;
         xSpare6 : Bool;
         xSpare7 : Bool;
         xSpare8 : Bool;
         xSpare9 : Bool;
         xSpare10 : Bool;   //
         xSpare11 : Bool;
         xSpare12 : Bool;
         xSpare13 : Bool;
         xSpare14 : Bool;
         xUpdateDistanceFromCenterLine : Bool;   // Bridge offset calibration request {x|x|x|x|M}
         xSpare16 : Bool;
         xSpare17 : Bool;
         xSpare18 : Bool;
         xSpare19 : Bool;
         xSpare20 : Bool;
         xSpare21 : Bool;
         xSpare22 : Bool;
         xSpare23 : Bool;
         xSpare24 : Bool;
         xSpare25 : Bool;
         xSpare26 : Bool;
         xSpare27 : Bool;
         xSpare28 : Bool;
         xSpare29 : Bool;
         xSpare30 : Bool;
         xSpare31 : Bool;
         xSpare : Array[0..15] of Bool;
         iSpare0 : Int;
         iSpare1 : Int;
         iSpare2 : Int;
         iSpare3 : Int;
         iSpare4 : Int;
         iSpare5 : Int;
         iSpare6 : Int;
         iSpare7 : Int;
         iSpare8 : Int;
         iSpare9 : Int;
         iSpare10 : Int;
         iSpare11 : Int;
         iSpare12 : Int;
         iSpare13 : Int;
         iSpare14 : Int;
         iSpare15 : Int;
         iSpare16 : Int;
         dDistanceFromCenterLine_cmm : DInt;   // Distance from center line {mm/100|mm|-3000|0|M}
         dSpare1 : DInt;   //
         dSpare2 : DInt;   //
         dSpare3 : DInt;
         dSpare4 : DInt;
         dSpare5 : DInt;
         dSpare6 : DInt;
         dSpare7 : DInt;
         dSpare8 : DInt;
         dSpare9 : DInt;
         dSpare10 : DInt;
         dSpare11 : DInt;
         dSpare12 : DInt;
         dSpare13 : DInt;
         dSpare14 : DInt;
         dSpare15 : DInt;
         dSpare16 : DInt;
         rSpare0 : Real;
         rSpare1 : Real;
         rSpare2 : Real;
         rSpare3 : Real;
         rSpare4 : Real;
         rSpare5 : Real;
         rSpare6 : Real;
         rSpare7 : Real;
         rSpare8 : Real;
         tManCmd : Struct
            xJogForward : Bool;   // Carriage manual jog forward {x|x|x|x|O}
            xJogBackward : Bool;   // Carriage manual jog backward {x|x|x|x|O}
            xSpare2 : Bool;
            xSpare3 : Bool;
            xSpare4 : Bool;
            xSpare5 : Bool;
            xSpare6 : Bool;
            xSpare7 : Bool;
            xSpare8 : Bool;
            xSpare9 : Bool;
            xSpare10 : Bool;
            xSpare11 : Bool;
            xSpare12 : Bool;
            xSpare13 : Bool;
            xSpare14 : Bool;
            xSpare15 : Bool;
            xSpare16 : Bool;
            xSpare17 : Bool;
            xSpare18 : Bool;
            xSpare19 : Bool;
            xSpare20 : Bool;
            xSpare21 : Bool;
            xSpare22 : Bool;
            xSpare23 : Bool;
            xSpare24 : Bool;
            xSpare25 : Bool;
            xSpare26 : Bool;
            xSpare27 : Bool;
            xSpare28 : Bool;
            xSpare29 : Bool;
            xSpare30 : Bool;
            xSpare31 : Bool;
         END_STRUCT;
      END_STRUCT;
   END_STRUCT;


BEGIN

END_DATA_BLOCK

DATA_BLOCK "DB_M220_2_HMI"
{ DB_Accessible_From_Webserver := 'FALSE' ;
 S7_Optimized_Access := 'FALSE' }
VERSION : 0.1
NON_RETAIN
   STRUCT
      tALM { ExternalWritable := 'False'} : Struct   // HMI Alarms
         tE { ExternalWritable := 'False'} : Struct   // Stopping faults
            xSpare_0 { ExternalWritable := 'False'} : Bool;
            xSpare_1 { ExternalWritable := 'False'} : Bool;
            xSpare_2 { ExternalWritable := 'False'} : Bool;
            xSpare_3 { ExternalWritable := 'False'} : Bool;
            xSpare_4 { ExternalWritable := 'False'} : Bool;
            xSpare_5 { ExternalWritable := 'False'} : Bool;
            xSpare_6 { ExternalWritable := 'False'} : Bool;
            xSpare_7 { ExternalWritable := 'False'} : Bool;
            xSpare_8 { ExternalWritable := 'False'} : Bool;
            xSpare_9 { ExternalWritable := 'False'} : Bool;
            xSpare_10 { ExternalWritable := 'False'} : Bool;
            xSpare_11 { ExternalWritable := 'False'} : Bool;
            xSpare_12 { ExternalWritable := 'False'} : Bool;
            xSpare_13 { ExternalWritable := 'False'} : Bool;
            xSpare_14 { ExternalWritable := 'False'} : Bool;
            xSpare_15 { ExternalWritable := 'False'} : Bool;
            xSpare_16 { ExternalWritable := 'False'} : Bool;
            xSpare_17 { ExternalWritable := 'False'} : Bool;
            xSpare_18 { ExternalWritable := 'False'} : Bool;
            xSpare_19 { ExternalWritable := 'False'} : Bool;
            xSpare_20 { ExternalWritable := 'False'} : Bool;
            xSpare_21 { ExternalWritable := 'False'} : Bool;
            xSpare_22 { ExternalWritable := 'False'} : Bool;
            xSpare_23 { ExternalWritable := 'False'} : Bool;
            xSpare_24 { ExternalWritable := 'False'} : Bool;
            xSpare_25 { ExternalWritable := 'False'} : Bool;
            xSpare_26 { ExternalWritable := 'False'} : Bool;
            xSpare_27 { ExternalWritable := 'False'} : Bool;
            xSpare_28 { ExternalWritable := 'False'} : Bool;
            xSpare_29 { ExternalWritable := 'False'} : Bool;
            xSpare_30 { ExternalWritable := 'False'} : Bool;
            xSpare_31 { ExternalWritable := 'False'} : Bool;
         END_STRUCT;
         tS { ExternalWritable := 'False'} : Struct
            x0 { ExternalWritable := 'False'} : Bool;   // AZ.Carriage homing timeout
            x1 { ExternalWritable := 'False'} : Bool;   // AZ.Carriage positioning timeout
            x2 { ExternalWritable := 'False'} : Bool;   // QM.Carriage translation overload cutout
            x3 { ExternalWritable := 'False'} : Bool;   // SQ.Forward overstroke translation
            x4 { ExternalWritable := 'False'} : Bool;   // SQ.Backward overstroke translation
            x5 { ExternalWritable := 'False'} : Bool;   // AZ.Feedback error
            x6 { ExternalWritable := 'False'} : Bool;   // AZ.Drive not enable
            x7 { ExternalWritable := 'False'} : Bool;   // AZ.Drive not ok
            x8 { ExternalWritable := 'False'} : Bool;   // AZ.Drive link timeout
            x9 { ExternalWritable := 'False'} : Bool;
            x10 { ExternalWritable := 'False'} : Bool;
            x11 { ExternalWritable := 'False'} : Bool;
            x12 { ExternalWritable := 'False'} : Bool;
            x13 { ExternalWritable := 'False'} : Bool;
            x14 { ExternalWritable := 'False'} : Bool;
            x15 { ExternalWritable := 'False'} : Bool;
            x16 { ExternalWritable := 'False'} : Bool;
            x17 { ExternalWritable := 'False'} : Bool;
            x18 { ExternalWritable := 'False'} : Bool;
            x19 { ExternalWritable := 'False'} : Bool;
            x20 { ExternalWritable := 'False'} : Bool;
            x21 { ExternalWritable := 'False'} : Bool;
            x22 { ExternalWritable := 'False'} : Bool;
            x23 { ExternalWritable := 'False'} : Bool;
            x24 { ExternalWritable := 'False'} : Bool;
            x25 { ExternalWritable := 'False'} : Bool;
            x26 { ExternalWritable := 'False'} : Bool;
            x27 { ExternalWritable := 'False'} : Bool;
            x28 { ExternalWritable := 'False'} : Bool;
            x29 { ExternalWritable := 'False'} : Bool;
            x30 { ExternalWritable := 'False'} : Bool;
            x31 { ExternalWritable := 'False'} : Bool;
         END_STRUCT;
         tF { ExternalAccessible := 'False'; ExternalVisible := 'False'; ExternalWritable := 'False'} : Struct   // Faults
            xSpare_0 { ExternalAccessible := 'False'; ExternalVisible := 'False'; ExternalWritable := 'False'} : Bool;
            xSpare_1 { ExternalAccessible := 'False'; ExternalVisible := 'False'; ExternalWritable := 'False'} : Bool;
            xSpare_2 { ExternalAccessible := 'False'; ExternalVisible := 'False'; ExternalWritable := 'False'} : Bool;
            xSpare_3 { ExternalAccessible := 'False'; ExternalVisible := 'False'; ExternalWritable := 'False'} : Bool;
            xSpare_4 { ExternalAccessible := 'False'; ExternalVisible := 'False'; ExternalWritable := 'False'} : Bool;
            xSpare_5 { ExternalAccessible := 'False'; ExternalVisible := 'False'; ExternalWritable := 'False'} : Bool;
            xSpare_6 { ExternalAccessible := 'False'; ExternalVisible := 'False'; ExternalWritable := 'False'} : Bool;
            xSpare_7 { ExternalAccessible := 'False'; ExternalVisible := 'False'; ExternalWritable := 'False'} : Bool;
            xSpare_8 { ExternalAccessible := 'False'; ExternalVisible := 'False'; ExternalWritable := 'False'} : Bool;
            xSpare_9 { ExternalAccessible := 'False'; ExternalVisible := 'False'; ExternalWritable := 'False'} : Bool;
            xSpare_10 { ExternalAccessible := 'False'; ExternalVisible := 'False'; ExternalWritable := 'False'} : Bool;
            xSpare_11 { ExternalAccessible := 'False'; ExternalVisible := 'False'; ExternalWritable := 'False'} : Bool;
            xSpare_12 { ExternalAccessible := 'False'; ExternalVisible := 'False'; ExternalWritable := 'False'} : Bool;
            xSpare_13 { ExternalAccessible := 'False'; ExternalVisible := 'False'; ExternalWritable := 'False'} : Bool;
            xSpare_14 { ExternalAccessible := 'False'; ExternalVisible := 'False'; ExternalWritable := 'False'} : Bool;
            xSpare_15 { ExternalAccessible := 'False'; ExternalVisible := 'False'; ExternalWritable := 'False'} : Bool;
            xSpare_16 { ExternalAccessible := 'False'; ExternalVisible := 'False'; ExternalWritable := 'False'} : Bool;
            xSpare_17 { ExternalAccessible := 'False'; ExternalVisible := 'False'; ExternalWritable := 'False'} : Bool;
            xSpare_18 { ExternalAccessible := 'False'; ExternalVisible := 'False'; ExternalWritable := 'False'} : Bool;
            xSpare_19 { ExternalAccessible := 'False'; ExternalVisible := 'False'; ExternalWritable := 'False'} : Bool;
            xSpare_20 { ExternalAccessible := 'False'; ExternalVisible := 'False'; ExternalWritable := 'False'} : Bool;
            xSpare_21 { ExternalAccessible := 'False'; ExternalVisible := 'False'; ExternalWritable := 'False'} : Bool;
            xSpare_22 { ExternalAccessible := 'False'; ExternalVisible := 'False'; ExternalWritable := 'False'} : Bool;
            xSpare_23 { ExternalAccessible := 'False'; ExternalVisible := 'False'; ExternalWritable := 'False'} : Bool;
            xSpare_24 { ExternalAccessible := 'False'; ExternalVisible := 'False'; ExternalWritable := 'False'} : Bool;
            xSpare_25 { ExternalAccessible := 'False'; ExternalVisible := 'False'; ExternalWritable := 'False'} : Bool;
            xSpare_26 { ExternalAccessible := 'False'; ExternalVisible := 'False'; ExternalWritable := 'False'} : Bool;
            xSpare_27 { ExternalAccessible := 'False'; ExternalVisible := 'False'; ExternalWritable := 'False'} : Bool;
            xSpare_28 { ExternalAccessible := 'False'; ExternalVisible := 'False'; ExternalWritable := 'False'} : Bool;
            xSpare_29 { ExternalAccessible := 'False'; ExternalVisible := 'False'; ExternalWritable := 'False'} : Bool;
            xSpare_30 { ExternalAccessible := 'False'; ExternalVisible := 'False'; ExternalWritable := 'False'} : Bool;
            xSpare_31 { ExternalAccessible := 'False'; ExternalVisible := 'False'; ExternalWritable := 'False'} : Bool;
         END_STRUCT;
         tW { ExternalAccessible := 'False'; ExternalVisible := 'False'; ExternalWritable := 'False'} : Struct   // Warnings
            xSpare_0 { ExternalAccessible := 'False'; ExternalVisible := 'False'; ExternalWritable := 'False'} : Bool;
            xSpare_1 { ExternalAccessible := 'False'; ExternalVisible := 'False'; ExternalWritable := 'False'} : Bool;
            xSpare_2 { ExternalAccessible := 'False'; ExternalVisible := 'False'; ExternalWritable := 'False'} : Bool;
            xSpare_3 { ExternalAccessible := 'False'; ExternalVisible := 'False'; ExternalWritable := 'False'} : Bool;
            xSpare_4 { ExternalAccessible := 'False'; ExternalVisible := 'False'; ExternalWritable := 'False'} : Bool;
            xSpare_5 { ExternalAccessible := 'False'; ExternalVisible := 'False'; ExternalWritable := 'False'} : Bool;
            xSpare_6 { ExternalAccessible := 'False'; ExternalVisible := 'False'; ExternalWritable := 'False'} : Bool;
            xSpare_7 { ExternalAccessible := 'False'; ExternalVisible := 'False'; ExternalWritable := 'False'} : Bool;
            xSpare_8 { ExternalAccessible := 'False'; ExternalVisible := 'False'; ExternalWritable := 'False'} : Bool;
            xSpare_9 { ExternalAccessible := 'False'; ExternalVisible := 'False'; ExternalWritable := 'False'} : Bool;
            xSpare_10 { ExternalAccessible := 'False'; ExternalVisible := 'False'; ExternalWritable := 'False'} : Bool;
            xSpare_11 { ExternalAccessible := 'False'; ExternalVisible := 'False'; ExternalWritable := 'False'} : Bool;
            xSpare_12 { ExternalAccessible := 'False'; ExternalVisible := 'False'; ExternalWritable := 'False'} : Bool;
            xSpare_13 { ExternalAccessible := 'False'; ExternalVisible := 'False'; ExternalWritable := 'False'} : Bool;
            xSpare_14 { ExternalAccessible := 'False'; ExternalVisible := 'False'; ExternalWritable := 'False'} : Bool;
            xSpare_15 { ExternalAccessible := 'False'; ExternalVisible := 'False'; ExternalWritable := 'False'} : Bool;
            xSpare_16 { ExternalAccessible := 'False'; ExternalVisible := 'False'; ExternalWritable := 'False'} : Bool;
            xSpare_17 { ExternalAccessible := 'False'; ExternalVisible := 'False'; ExternalWritable := 'False'} : Bool;
            xSpare_18 { ExternalAccessible := 'False'; ExternalVisible := 'False'; ExternalWritable := 'False'} : Bool;
            xSpare_19 { ExternalAccessible := 'False'; ExternalVisible := 'False'; ExternalWritable := 'False'} : Bool;
            xSpare_20 { ExternalAccessible := 'False'; ExternalVisible := 'False'; ExternalWritable := 'False'} : Bool;
            xSpare_21 { ExternalAccessible := 'False'; ExternalVisible := 'False'; ExternalWritable := 'False'} : Bool;
            xSpare_22 { ExternalAccessible := 'False'; ExternalVisible := 'False'; ExternalWritable := 'False'} : Bool;
            xSpare_23 { ExternalAccessible := 'False'; ExternalVisible := 'False'; ExternalWritable := 'False'} : Bool;
            xSpare_24 { ExternalAccessible := 'False'; ExternalVisible := 'False'; ExternalWritable := 'False'} : Bool;
            xSpare_25 { ExternalAccessible := 'False'; ExternalVisible := 'False'; ExternalWritable := 'False'} : Bool;
            xSpare_26 { ExternalAccessible := 'False'; ExternalVisible := 'False'; ExternalWritable := 'False'} : Bool;
            xSpare_27 { ExternalAccessible := 'False'; ExternalVisible := 'False'; ExternalWritable := 'False'} : Bool;
            xSpare_28 { ExternalAccessible := 'False'; ExternalVisible := 'False'; ExternalWritable := 'False'} : Bool;
            xSpare_29 { ExternalAccessible := 'False'; ExternalVisible := 'False'; ExternalWritable := 'False'} : Bool;
            xSpare_30 { ExternalAccessible := 'False'; ExternalVisible := 'False'; ExternalWritable := 'False'} : Bool;
            xSpare_31 { ExternalAccessible := 'False'; ExternalVisible := 'False'; ExternalWritable := 'False'} : Bool;
         END_STRUCT;
      END_STRUCT;
      tHMR { ExternalWritable := 'False'} : Struct   // HMI Read
         xCalibrationsAllowed { ExternalWritable := 'False'} : Bool;   // Calibrations allowed {x|x|x|x|O}
         xSpare1 { ExternalWritable := 'False'} : Bool;
         xSpare2 { ExternalWritable := 'False'} : Bool;
         xSpare3 { ExternalWritable := 'False'} : Bool;
         xSpare4 { ExternalWritable := 'False'} : Bool;
         xSpare5 { ExternalWritable := 'False'} : Bool;
         xSpare6 { ExternalWritable := 'False'} : Bool;
         xSpare7 { ExternalWritable := 'False'} : Bool;
         xSpare8 { ExternalWritable := 'False'} : Bool;
         xSpare9 { ExternalWritable := 'False'} : Bool;
         xSpare10 { ExternalWritable := 'False'} : Bool;
         xSpare11 { ExternalWritable := 'False'} : Bool;
         xSpare12 { ExternalWritable := 'False'} : Bool;
         xSpare13 { ExternalWritable := 'False'} : Bool;
         xSpare14 { ExternalWritable := 'False'} : Bool;   //
         xSpare15 { ExternalWritable := 'False'} : Bool;
         xSpare16 { ExternalWritable := 'False'} : Bool;
         xSpare17 { ExternalWritable := 'False'} : Bool;
         xSpare18 { ExternalWritable := 'False'} : Bool;
         xSpare19 { ExternalWritable := 'False'} : Bool;
         xSpare20 { ExternalWritable := 'False'} : Bool;
         xSpare21 { ExternalWritable := 'False'} : Bool;
         xSpare22 { ExternalWritable := 'False'} : Bool;
         xSpare23 { ExternalWritable := 'False'} : Bool;
         xSpare24 { ExternalWritable := 'False'} : Bool;
         xSpare25 { ExternalWritable := 'False'} : Bool;
         xSpare26 { ExternalWritable := 'False'} : Bool;
         xSpare27 { ExternalWritable := 'False'} : Bool;
         xSpare28 { ExternalWritable := 'False'} : Bool;
         xSpare29 { ExternalWritable := 'False'} : Bool;
         xSpare30 { ExternalWritable := 'False'} : Bool;
         xSpare31 { ExternalWritable := 'False'} : Bool;
         xSpare { ExternalWritable := 'False'} : Array[0..15] of Bool;
         iSpare0 { ExternalWritable := 'False'} : Int;
         iSpare1 { ExternalWritable := 'False'} : Int;
         iSpare2 { ExternalWritable := 'False'} : Int;
         iSpare3 { ExternalWritable := 'False'} : Int;
         iSpare4 { ExternalWritable := 'False'} : Int;
         iSpare5 { ExternalWritable := 'False'} : Int;
         iSpare6 { ExternalWritable := 'False'} : Int;
         iSpare7 { ExternalWritable := 'False'} : Int;
         iSpare8 { ExternalWritable := 'False'} : Int;
         iSpare9 { ExternalWritable := 'False'} : Int;
         iSpare10 { ExternalWritable := 'False'} : Int;
         iSpare11 { ExternalWritable := 'False'} : Int;
         iSpare12 { ExternalWritable := 'False'} : Int;
         iSpare13 { ExternalWritable := 'False'} : Int;
         iSpare14 { ExternalWritable := 'False'} : Int;
         iSpare15 { ExternalWritable := 'False'} : Int;
         iSpare16 { ExternalWritable := 'False'} : Int;
         dCarriageStatus { ExternalWritable := 'False'} : DInt;   // Carriage status (1=Not Initialized 2=Not referred 3=Not positioned 4=Positioned 5=Positioning 6=Virtual collision 7=Anomaly) {x|x|x|x|O}
         dCarriageHomePosition_cmm { ExternalWritable := 'False'} : DInt;   // Carriage home position [mm/100] {mm/100|mm|x|x|O}
         dCarriageActualPosition_cmm { ExternalWritable := 'False'} : DInt;   // Carriage actual position [mm/100] {mm/100|mm|x|x|O}
         dSpare3 { ExternalWritable := 'False'} : DInt;
         dSpare4 { ExternalWritable := 'False'} : DInt;
         dSpare5 { ExternalWritable := 'False'} : DInt;
         dSpare6 { ExternalWritable := 'False'} : DInt;
         dSpare7 { ExternalWritable := 'False'} : DInt;
         dSpare8 { ExternalWritable := 'False'} : DInt;
         dSpare9 { ExternalWritable := 'False'} : DInt;
         dSpare10 { ExternalWritable := 'False'} : DInt;
         dSpare11 { ExternalWritable := 'False'} : DInt;
         dSpare12 { ExternalWritable := 'False'} : DInt;
         dSpare13 { ExternalWritable := 'False'} : DInt;
         dSpare14 { ExternalWritable := 'False'} : DInt;
         dSpare15 { ExternalWritable := 'False'} : DInt;
         rSpare0 { ExternalWritable := 'False'} : Real;
         rSpare1 { ExternalWritable := 'False'} : Real;
         rSpare2 { ExternalWritable := 'False'} : Real;
         rSpare3 { ExternalWritable := 'False'} : Real;
         rSpare4 { ExternalWritable := 'False'} : Real;
         rSpare5 { ExternalWritable := 'False'} : Real;
         rSpare6 { ExternalWritable := 'False'} : Real;
         rSpare7 { ExternalWritable := 'False'} : Real;
         rSpare8 { ExternalWritable := 'False'} : Real;
         tManCmd { ExternalWritable := 'False'} : Struct
            xJogForward { ExternalWritable := 'False'} : Bool;   // Carriage manual jog forward fdbk {x|x|x|x|O}
            xJogBackward { ExternalWritable := 'False'} : Bool;   // Carriage manual jog backward fdbk {x|x|x|x|O}
            xSpare2 { ExternalWritable := 'False'} : Bool;
            xSpare3 { ExternalWritable := 'False'} : Bool;
            xSpare4 { ExternalWritable := 'False'} : Bool;
            xSpare5 { ExternalWritable := 'False'} : Bool;
            xSpare6 { ExternalWritable := 'False'} : Bool;
            xSpare7 { ExternalWritable := 'False'} : Bool;
            xSpare8 { ExternalWritable := 'False'} : Bool;
            xSpare9 { ExternalWritable := 'False'} : Bool;
            xSpare10 { ExternalWritable := 'False'} : Bool;
            xSpare11 { ExternalWritable := 'False'} : Bool;
            xSpare12 { ExternalWritable := 'False'} : Bool;
            xSpare13 { ExternalWritable := 'False'} : Bool;
            xSpare14 { ExternalWritable := 'False'} : Bool;
            xSpare15 { ExternalWritable := 'False'} : Bool;
            xSpare { ExternalWritable := 'False'} : Array[0..15] of Bool;
         END_STRUCT;
      END_STRUCT;
      tHMW : Struct   // HMI Write
         xForceCarriageHoming : Bool;   // Force the homing of the carriage {x|x|x|x|M}
         xSpare1 : Bool;
         xSpare2 : Bool;
         xSpare3 : Bool;
         xSpare4 : Bool;
         xSpare5 : Bool;
         xSpare6 : Bool;
         xSpare7 : Bool;
         xSpare8 : Bool;
         xSpare9 : Bool;
         xSpare10 : Bool;   //
         xSpare11 : Bool;
         xSpare12 : Bool;
         xSpare13 : Bool;
         xSpare14 : Bool;
         xUpdateDistanceFromCenterLine : Bool;   // Bridge offset calibration request {x|x|x|x|M}
         xSpare16 : Bool;
         xSpare17 : Bool;
         xSpare18 : Bool;
         xSpare19 : Bool;
         xSpare20 : Bool;
         xSpare21 : Bool;
         xSpare22 : Bool;
         xSpare23 : Bool;
         xSpare24 : Bool;
         xSpare25 : Bool;
         xSpare26 : Bool;
         xSpare27 : Bool;
         xSpare28 : Bool;
         xSpare29 : Bool;
         xSpare30 : Bool;
         xSpare31 : Bool;
         xSpare : Array[0..15] of Bool;
         iSpare0 : Int;
         iSpare1 : Int;
         iSpare2 : Int;
         iSpare3 : Int;
         iSpare4 : Int;
         iSpare5 : Int;
         iSpare6 : Int;
         iSpare7 : Int;
         iSpare8 : Int;
         iSpare9 : Int;
         iSpare10 : Int;
         iSpare11 : Int;
         iSpare12 : Int;
         iSpare13 : Int;
         iSpare14 : Int;
         iSpare15 : Int;
         iSpare16 : Int;
         dDistanceFromCenterLine_cmm : DInt;   // Distance from center line {mm/100|mm|-3000|0|M}
         dSpare1 : DInt;   //
         dSpare2 : DInt;   //
         dSpare3 : DInt;
         dSpare4 : DInt;
         dSpare5 : DInt;
         dSpare6 : DInt;
         dSpare7 : DInt;
         dSpare8 : DInt;
         dSpare9 : DInt;
         dSpare10 : DInt;
         dSpare11 : DInt;
         dSpare12 : DInt;
         dSpare13 : DInt;
         dSpare14 : DInt;
         dSpare15 : DInt;
         dSpare16 : DInt;
         rSpare0 : Real;
         rSpare1 : Real;
         rSpare2 : Real;
         rSpare3 : Real;
         rSpare4 : Real;
         rSpare5 : Real;
         rSpare6 : Real;
         rSpare7 : Real;
         rSpare8 : Real;
         tManCmd : Struct
            xJogForward : Bool;   // Carriage manual jog forward {x|x|x|x|O}
            xJogBackward : Bool;   // Carriage manual jog backward {x|x|x|x|O}
            xSpare2 { ExternalWritable := 'False'} : Bool;
            xSpare3 { ExternalWritable := 'False'} : Bool;
            xSpare4 { ExternalWritable := 'False'} : Bool;
            xSpare5 { ExternalWritable := 'False'} : Bool;
            xSpare6 { ExternalWritable := 'False'} : Bool;
            xSpare7 { ExternalWritable := 'False'} : Bool;
            xSpare8 { ExternalWritable := 'False'} : Bool;
            xSpare9 { ExternalWritable := 'False'} : Bool;
            xSpare10 { ExternalWritable := 'False'} : Bool;
            xSpare11 { ExternalWritable := 'False'} : Bool;
            xSpare12 { ExternalWritable := 'False'} : Bool;
            xSpare13 { ExternalWritable := 'False'} : Bool;
            xSpare14 { ExternalWritable := 'False'} : Bool;
            xSpare15 { ExternalWritable := 'False'} : Bool;
            xSpare16 : Bool;
            xSpare17 : Bool;
            xSpare18 : Bool;
            xSpare19 : Bool;
            xSpare20 : Bool;
            xSpare21 : Bool;
            xSpare22 : Bool;
            xSpare23 : Bool;
            xSpare24 : Bool;
            xSpare25 : Bool;
            xSpare26 : Bool;
            xSpare27 : Bool;
            xSpare28 : Bool;
            xSpare29 : Bool;
            xSpare30 : Bool;
            xSpare31 : Bool;
         END_STRUCT;
      END_STRUCT;
   END_STRUCT;


BEGIN

END_DATA_BLOCK

DATA_BLOCK "DB_M220_1_HMI"
{ DB_Accessible_From_Webserver := 'FALSE' ;
 S7_Optimized_Access := 'FALSE' }
VERSION : 0.1
NON_RETAIN
   STRUCT
      tALM { ExternalWritable := 'False'} : Struct   // HMI Alarms
         tE { ExternalWritable := 'False'} : Struct   // Stopping faults
            xSpare_0 { ExternalWritable := 'False'} : Bool;
            xSpare_1 { ExternalWritable := 'False'} : Bool;
            xSpare_2 { ExternalWritable := 'False'} : Bool;
            xSpare_3 { ExternalWritable := 'False'} : Bool;
            xSpare_4 { ExternalWritable := 'False'} : Bool;
            xSpare_5 { ExternalWritable := 'False'} : Bool;
            xSpare_6 { ExternalWritable := 'False'} : Bool;
            xSpare_7 { ExternalWritable := 'False'} : Bool;
            xSpare_8 { ExternalWritable := 'False'} : Bool;
            xSpare_9 { ExternalWritable := 'False'} : Bool;
            xSpare_10 { ExternalWritable := 'False'} : Bool;
            xSpare_11 { ExternalWritable := 'False'} : Bool;
            xSpare_12 { ExternalWritable := 'False'} : Bool;
            xSpare_13 { ExternalWritable := 'False'} : Bool;
            xSpare_14 { ExternalWritable := 'False'} : Bool;
            xSpare_15 { ExternalWritable := 'False'} : Bool;
            xSpare_16 { ExternalWritable := 'False'} : Bool;
            xSpare_17 { ExternalWritable := 'False'} : Bool;
            xSpare_18 { ExternalWritable := 'False'} : Bool;
            xSpare_19 { ExternalWritable := 'False'} : Bool;
            xSpare_20 { ExternalWritable := 'False'} : Bool;
            xSpare_21 { ExternalWritable := 'False'} : Bool;
            xSpare_22 { ExternalWritable := 'False'} : Bool;
            xSpare_23 { ExternalWritable := 'False'} : Bool;
            xSpare_24 { ExternalWritable := 'False'} : Bool;
            xSpare_25 { ExternalWritable := 'False'} : Bool;
            xSpare_26 { ExternalWritable := 'False'} : Bool;
            xSpare_27 { ExternalWritable := 'False'} : Bool;
            xSpare_28 { ExternalWritable := 'False'} : Bool;
            xSpare_29 { ExternalWritable := 'False'} : Bool;
            xSpare_30 { ExternalWritable := 'False'} : Bool;
            xSpare_31 { ExternalWritable := 'False'} : Bool;
         END_STRUCT;
         tS { ExternalWritable := 'False'} : Struct
            x0 { ExternalWritable := 'False'} : Bool;   // AZ.Carriage homing timeout
            x1 { ExternalWritable := 'False'} : Bool;   // AZ.Carriage positioning timeout
            x2 { ExternalWritable := 'False'} : Bool;   // QM.Carriage translation overload cutout
            x3 { ExternalWritable := 'False'} : Bool;   // SQ.Forward overstroke translation
            x4 { ExternalWritable := 'False'} : Bool;   // SQ.Backward overstroke translation
            x5 { ExternalWritable := 'False'} : Bool;   // AZ.Feedback error
            x6 { ExternalWritable := 'False'} : Bool;   // AZ.Drive not enable
            x7 { ExternalWritable := 'False'} : Bool;   // AZ.Drive not ok
            x8 { ExternalWritable := 'False'} : Bool;   // AZ.Drive link timeout
            x9 { ExternalWritable := 'False'} : Bool;
            x10 { ExternalWritable := 'False'} : Bool;
            x11 { ExternalWritable := 'False'} : Bool;
            x12 { ExternalWritable := 'False'} : Bool;
            x13 { ExternalWritable := 'False'} : Bool;
            x14 { ExternalWritable := 'False'} : Bool;
            x15 { ExternalWritable := 'False'} : Bool;
            x16 { ExternalWritable := 'False'} : Bool;
            x17 { ExternalWritable := 'False'} : Bool;
            x18 { ExternalWritable := 'False'} : Bool;
            x19 { ExternalWritable := 'False'} : Bool;
            x20 { ExternalWritable := 'False'} : Bool;
            x21 { ExternalWritable := 'False'} : Bool;
            x22 { ExternalWritable := 'False'} : Bool;
            x23 { ExternalWritable := 'False'} : Bool;
            x24 { ExternalWritable := 'False'} : Bool;
            x25 { ExternalWritable := 'False'} : Bool;
            x26 { ExternalWritable := 'False'} : Bool;
            x27 { ExternalWritable := 'False'} : Bool;
            x28 { ExternalWritable := 'False'} : Bool;
            x29 { ExternalWritable := 'False'} : Bool;
            x30 { ExternalWritable := 'False'} : Bool;
            x31 { ExternalWritable := 'False'} : Bool;
         END_STRUCT;
         tF { ExternalAccessible := 'False'; ExternalVisible := 'False'; ExternalWritable := 'False'} : Struct   // Faults
            xSpare_0 { ExternalAccessible := 'False'; ExternalVisible := 'False'; ExternalWritable := 'False'} : Bool;
            xSpare_1 { ExternalAccessible := 'False'; ExternalVisible := 'False'; ExternalWritable := 'False'} : Bool;
            xSpare_2 { ExternalAccessible := 'False'; ExternalVisible := 'False'; ExternalWritable := 'False'} : Bool;
            xSpare_3 { ExternalAccessible := 'False'; ExternalVisible := 'False'; ExternalWritable := 'False'} : Bool;
            xSpare_4 { ExternalAccessible := 'False'; ExternalVisible := 'False'; ExternalWritable := 'False'} : Bool;
            xSpare_5 { ExternalAccessible := 'False'; ExternalVisible := 'False'; ExternalWritable := 'False'} : Bool;
            xSpare_6 { ExternalAccessible := 'False'; ExternalVisible := 'False'; ExternalWritable := 'False'} : Bool;
            xSpare_7 { ExternalAccessible := 'False'; ExternalVisible := 'False'; ExternalWritable := 'False'} : Bool;
            xSpare_8 { ExternalAccessible := 'False'; ExternalVisible := 'False'; ExternalWritable := 'False'} : Bool;
            xSpare_9 { ExternalAccessible := 'False'; ExternalVisible := 'False'; ExternalWritable := 'False'} : Bool;
            xSpare_10 { ExternalAccessible := 'False'; ExternalVisible := 'False'; ExternalWritable := 'False'} : Bool;
            xSpare_11 { ExternalAccessible := 'False'; ExternalVisible := 'False'; ExternalWritable := 'False'} : Bool;
            xSpare_12 { ExternalAccessible := 'False'; ExternalVisible := 'False'; ExternalWritable := 'False'} : Bool;
            xSpare_13 { ExternalAccessible := 'False'; ExternalVisible := 'False'; ExternalWritable := 'False'} : Bool;
            xSpare_14 { ExternalAccessible := 'False'; ExternalVisible := 'False'; ExternalWritable := 'False'} : Bool;
            xSpare_15 { ExternalAccessible := 'False'; ExternalVisible := 'False'; ExternalWritable := 'False'} : Bool;
            xSpare_16 { ExternalAccessible := 'False'; ExternalVisible := 'False'; ExternalWritable := 'False'} : Bool;
            xSpare_17 { ExternalAccessible := 'False'; ExternalVisible := 'False'; ExternalWritable := 'False'} : Bool;
            xSpare_18 { ExternalAccessible := 'False'; ExternalVisible := 'False'; ExternalWritable := 'False'} : Bool;
            xSpare_19 { ExternalAccessible := 'False'; ExternalVisible := 'False'; ExternalWritable := 'False'} : Bool;
            xSpare_20 { ExternalAccessible := 'False'; ExternalVisible := 'False'; ExternalWritable := 'False'} : Bool;
            xSpare_21 { ExternalAccessible := 'False'; ExternalVisible := 'False'; ExternalWritable := 'False'} : Bool;
            xSpare_22 { ExternalAccessible := 'False'; ExternalVisible := 'False'; ExternalWritable := 'False'} : Bool;
            xSpare_23 { ExternalAccessible := 'False'; ExternalVisible := 'False'; ExternalWritable := 'False'} : Bool;
            xSpare_24 { ExternalAccessible := 'False'; ExternalVisible := 'False'; ExternalWritable := 'False'} : Bool;
            xSpare_25 { ExternalAccessible := 'False'; ExternalVisible := 'False'; ExternalWritable := 'False'} : Bool;
            xSpare_26 { ExternalAccessible := 'False'; ExternalVisible := 'False'; ExternalWritable := 'False'} : Bool;
            xSpare_27 { ExternalAccessible := 'False'; ExternalVisible := 'False'; ExternalWritable := 'False'} : Bool;
            xSpare_28 { ExternalAccessible := 'False'; ExternalVisible := 'False'; ExternalWritable := 'False'} : Bool;
            xSpare_29 { ExternalAccessible := 'False'; ExternalVisible := 'False'; ExternalWritable := 'False'} : Bool;
            xSpare_30 { ExternalAccessible := 'False'; ExternalVisible := 'False'; ExternalWritable := 'False'} : Bool;
            xSpare_31 { ExternalAccessible := 'False'; ExternalVisible := 'False'; ExternalWritable := 'False'} : Bool;
         END_STRUCT;
         tW { ExternalAccessible := 'False'; ExternalVisible := 'False'; ExternalWritable := 'False'} : Struct   // Warnings
            xSpare_0 { ExternalAccessible := 'False'; ExternalVisible := 'False'; ExternalWritable := 'False'} : Bool;
            xSpare_1 { ExternalAccessible := 'False'; ExternalVisible := 'False'; ExternalWritable := 'False'} : Bool;
            xSpare_2 { ExternalAccessible := 'False'; ExternalVisible := 'False'; ExternalWritable := 'False'} : Bool;
            xSpare_3 { ExternalAccessible := 'False'; ExternalVisible := 'False'; ExternalWritable := 'False'} : Bool;
            xSpare_4 { ExternalAccessible := 'False'; ExternalVisible := 'False'; ExternalWritable := 'False'} : Bool;
            xSpare_5 { ExternalAccessible := 'False'; ExternalVisible := 'False'; ExternalWritable := 'False'} : Bool;
            xSpare_6 { ExternalAccessible := 'False'; ExternalVisible := 'False'; ExternalWritable := 'False'} : Bool;
            xSpare_7 { ExternalAccessible := 'False'; ExternalVisible := 'False'; ExternalWritable := 'False'} : Bool;
            xSpare_8 { ExternalAccessible := 'False'; ExternalVisible := 'False'; ExternalWritable := 'False'} : Bool;
            xSpare_9 { ExternalAccessible := 'False'; ExternalVisible := 'False'; ExternalWritable := 'False'} : Bool;
            xSpare_10 { ExternalAccessible := 'False'; ExternalVisible := 'False'; ExternalWritable := 'False'} : Bool;
            xSpare_11 { ExternalAccessible := 'False'; ExternalVisible := 'False'; ExternalWritable := 'False'} : Bool;
            xSpare_12 { ExternalAccessible := 'False'; ExternalVisible := 'False'; ExternalWritable := 'False'} : Bool;
            xSpare_13 { ExternalAccessible := 'False'; ExternalVisible := 'False'; ExternalWritable := 'False'} : Bool;
            xSpare_14 { ExternalAccessible := 'False'; ExternalVisible := 'False'; ExternalWritable := 'False'} : Bool;
            xSpare_15 { ExternalAccessible := 'False'; ExternalVisible := 'False'; ExternalWritable := 'False'} : Bool;
            xSpare_16 { ExternalAccessible := 'False'; ExternalVisible := 'False'; ExternalWritable := 'False'} : Bool;
            xSpare_17 { ExternalAccessible := 'False'; ExternalVisible := 'False'; ExternalWritable := 'False'} : Bool;
            xSpare_18 { ExternalAccessible := 'False'; ExternalVisible := 'False'; ExternalWritable := 'False'} : Bool;
            xSpare_19 { ExternalAccessible := 'False'; ExternalVisible := 'False'; ExternalWritable := 'False'} : Bool;
            xSpare_20 { ExternalAccessible := 'False'; ExternalVisible := 'False'; ExternalWritable := 'False'} : Bool;
            xSpare_21 { ExternalAccessible := 'False'; ExternalVisible := 'False'; ExternalWritable := 'False'} : Bool;
            xSpare_22 { ExternalAccessible := 'False'; ExternalVisible := 'False'; ExternalWritable := 'False'} : Bool;
            xSpare_23 { ExternalAccessible := 'False'; ExternalVisible := 'False'; ExternalWritable := 'False'} : Bool;
            xSpare_24 { ExternalAccessible := 'False'; ExternalVisible := 'False'; ExternalWritable := 'False'} : Bool;
            xSpare_25 { ExternalAccessible := 'False'; ExternalVisible := 'False'; ExternalWritable := 'False'} : Bool;
            xSpare_26 { ExternalAccessible := 'False'; ExternalVisible := 'False'; ExternalWritable := 'False'} : Bool;
            xSpare_27 { ExternalAccessible := 'False'; ExternalVisible := 'False'; ExternalWritable := 'False'} : Bool;
            xSpare_28 { ExternalAccessible := 'False'; ExternalVisible := 'False'; ExternalWritable := 'False'} : Bool;
            xSpare_29 { ExternalAccessible := 'False'; ExternalVisible := 'False'; ExternalWritable := 'False'} : Bool;
            xSpare_30 { ExternalAccessible := 'False'; ExternalVisible := 'False'; ExternalWritable := 'False'} : Bool;
            xSpare_31 { ExternalAccessible := 'False'; ExternalVisible := 'False'; ExternalWritable := 'False'} : Bool;
         END_STRUCT;
      END_STRUCT;
      tHMR { ExternalWritable := 'False'} : Struct   // HMI Read
         xCalibrationsAllowed { ExternalWritable := 'False'} : Bool;   // Calibrations allowed {x|x|x|x|O}
         xSpare1 { ExternalWritable := 'False'} : Bool;
         xSpare2 { ExternalWritable := 'False'} : Bool;
         xSpare3 { ExternalWritable := 'False'} : Bool;
         xSpare4 { ExternalWritable := 'False'} : Bool;
         xSpare5 { ExternalWritable := 'False'} : Bool;
         xSpare6 { ExternalWritable := 'False'} : Bool;
         xSpare7 { ExternalWritable := 'False'} : Bool;
         xSpare8 { ExternalWritable := 'False'} : Bool;
         xSpare9 { ExternalWritable := 'False'} : Bool;
         xSpare10 { ExternalWritable := 'False'} : Bool;
         xSpare11 { ExternalWritable := 'False'} : Bool;
         xSpare12 { ExternalWritable := 'False'} : Bool;
         xSpare13 { ExternalWritable := 'False'} : Bool;
         xSpare14 { ExternalWritable := 'False'} : Bool;   //
         xSpare15 { ExternalWritable := 'False'} : Bool;
         xSpare16 { ExternalWritable := 'False'} : Bool;
         xSpare17 { ExternalWritable := 'False'} : Bool;
         xSpare18 { ExternalWritable := 'False'} : Bool;
         xSpare19 { ExternalWritable := 'False'} : Bool;
         xSpare20 { ExternalWritable := 'False'} : Bool;
         xSpare21 { ExternalWritable := 'False'} : Bool;
         xSpare22 { ExternalWritable := 'False'} : Bool;
         xSpare23 { ExternalWritable := 'False'} : Bool;
         xSpare24 { ExternalWritable := 'False'} : Bool;
         xSpare25 { ExternalWritable := 'False'} : Bool;
         xSpare26 { ExternalWritable := 'False'} : Bool;
         xSpare27 { ExternalWritable := 'False'} : Bool;
         xSpare28 { ExternalWritable := 'False'} : Bool;
         xSpare29 { ExternalWritable := 'False'} : Bool;
         xSpare30 { ExternalWritable := 'False'} : Bool;
         xSpare31 { ExternalWritable := 'False'} : Bool;
         xSpare { ExternalWritable := 'False'} : Array[0..15] of Bool;
         iSpare0 { ExternalWritable := 'False'} : Int;
         iSpare1 { ExternalWritable := 'False'} : Int;
         iSpare2 { ExternalWritable := 'False'} : Int;
         iSpare3 { ExternalWritable := 'False'} : Int;
         iSpare4 { ExternalWritable := 'False'} : Int;
         iSpare5 { ExternalWritable := 'False'} : Int;
         iSpare6 { ExternalWritable := 'False'} : Int;
         iSpare7 { ExternalWritable := 'False'} : Int;
         iSpare8 { ExternalWritable := 'False'} : Int;
         iSpare9 { ExternalWritable := 'False'} : Int;
         iSpare10 { ExternalWritable := 'False'} : Int;
         iSpare11 { ExternalWritable := 'False'} : Int;
         iSpare12 { ExternalWritable := 'False'} : Int;
         iSpare13 { ExternalWritable := 'False'} : Int;
         iSpare14 { ExternalWritable := 'False'} : Int;
         iSpare15 { ExternalWritable := 'False'} : Int;
         iSpare16 { ExternalWritable := 'False'} : Int;
         dCarriageStatus { ExternalWritable := 'False'} : DInt;   // Carriage status (1=Not Initialized 2=Not referred 3=Not positioned 4=Positioned 5=Positioning 6=Virtual collision 7=Anomaly) {x|x|x|x|O}
         dCarriageHomePosition_cmm { ExternalWritable := 'False'} : DInt;   // Carriage home position [mm/100] {mm/100|mm|x|x|O}
         dCarriageActualPosition_cmm { ExternalWritable := 'False'} : DInt;   // Carriage actual position [mm/100] {mm/100|mm|x|x|O}
         dSpare3 { ExternalWritable := 'False'} : DInt;
         dSpare4 { ExternalWritable := 'False'} : DInt;
         dSpare5 { ExternalWritable := 'False'} : DInt;
         dSpare6 { ExternalWritable := 'False'} : DInt;
         dSpare7 { ExternalWritable := 'False'} : DInt;
         dSpare8 { ExternalWritable := 'False'} : DInt;
         dSpare9 { ExternalWritable := 'False'} : DInt;
         dSpare10 { ExternalWritable := 'False'} : DInt;
         dSpare11 { ExternalWritable := 'False'} : DInt;
         dSpare12 { ExternalWritable := 'False'} : DInt;
         dSpare13 { ExternalWritable := 'False'} : DInt;
         dSpare14 { ExternalWritable := 'False'} : DInt;
         dSpare15 { ExternalWritable := 'False'} : DInt;
         rSpare0 { ExternalWritable := 'False'} : Real;
         rSpare1 { ExternalWritable := 'False'} : Real;
         rSpare2 { ExternalWritable := 'False'} : Real;
         rSpare3 { ExternalWritable := 'False'} : Real;
         rSpare4 { ExternalWritable := 'False'} : Real;
         rSpare5 { ExternalWritable := 'False'} : Real;
         rSpare6 { ExternalWritable := 'False'} : Real;
         rSpare7 { ExternalWritable := 'False'} : Real;
         rSpare8 { ExternalWritable := 'False'} : Real;
         tManCmd { ExternalWritable := 'False'} : Struct
            xJogForward { ExternalWritable := 'False'} : Bool;   // Carriage manual jog forward fdbk {x|x|x|x|O}
            xJogBackward { ExternalWritable := 'False'} : Bool;   // Carriage manual jog backward fdbk {x|x|x|x|O}
            xSpare2 { ExternalWritable := 'False'} : Bool;
            xSpare3 { ExternalWritable := 'False'} : Bool;
            xSpare4 { ExternalWritable := 'False'} : Bool;
            xSpare5 { ExternalWritable := 'False'} : Bool;
            xSpare6 { ExternalWritable := 'False'} : Bool;
            xSpare7 { ExternalWritable := 'False'} : Bool;
            xSpare8 { ExternalWritable := 'False'} : Bool;
            xSpare9 { ExternalWritable := 'False'} : Bool;
            xSpare10 { ExternalWritable := 'False'} : Bool;
            xSpare11 { ExternalWritable := 'False'} : Bool;
            xSpare12 { ExternalWritable := 'False'} : Bool;
            xSpare13 { ExternalWritable := 'False'} : Bool;
            xSpare14 { ExternalWritable := 'False'} : Bool;
            xSpare15 { ExternalWritable := 'False'} : Bool;
            xSpare { ExternalWritable := 'False'} : Array[0..15] of Bool;
         END_STRUCT;
      END_STRUCT;
      tHMW : Struct   // HMI Write
         xForceCarriageHoming : Bool;   // Force the homing of the carriage {x|x|x|x|M}
         xSpare1 : Bool;
         xSpare2 : Bool;
         xSpare3 : Bool;
         xSpare4 : Bool;
         xSpare5 : Bool;
         xSpare6 : Bool;
         xSpare7 : Bool;
         xSpare8 : Bool;
         xSpare9 : Bool;
         xSpare10 : Bool;   //
         xSpare11 : Bool;
         xSpare12 : Bool;
         xSpare13 : Bool;
         xSpare14 : Bool;
         xUpdateDistanceFromCenterLine : Bool;   // Bridge offset calibration request {x|x|x|x|M}
         xSpare16 : Bool;
         xSpare17 : Bool;
         xSpare18 : Bool;
         xSpare19 : Bool;
         xSpare20 : Bool;
         xSpare21 : Bool;
         xSpare22 : Bool;
         xSpare23 : Bool;
         xSpare24 : Bool;
         xSpare25 : Bool;
         xSpare26 : Bool;
         xSpare27 : Bool;
         xSpare28 : Bool;
         xSpare29 : Bool;
         xSpare30 : Bool;
         xSpare31 : Bool;
         xSpare : Array[0..15] of Bool;
         iSpare0 : Int;
         iSpare1 : Int;
         iSpare2 : Int;
         iSpare3 : Int;
         iSpare4 : Int;
         iSpare5 : Int;
         iSpare6 : Int;
         iSpare7 : Int;
         iSpare8 : Int;
         iSpare9 : Int;
         iSpare10 : Int;
         iSpare11 : Int;
         iSpare12 : Int;
         iSpare13 : Int;
         iSpare14 : Int;
         iSpare15 : Int;
         iSpare16 : Int;
         dDistanceFromCenterLine_cmm : DInt;   // Distance from center line {mm/100|mm|-3000|0|M}
         dSpare1 : DInt;   //
         dSpare2 : DInt;   //
         dSpare3 : DInt;
         dSpare4 : DInt;
         dSpare5 : DInt;
         dSpare6 : DInt;
         dSpare7 : DInt;
         dSpare8 : DInt;
         dSpare9 : DInt;
         dSpare10 : DInt;
         dSpare11 : DInt;
         dSpare12 : DInt;
         dSpare13 : DInt;
         dSpare14 : DInt;
         dSpare15 : DInt;
         dSpare16 : DInt;
         rSpare0 : Real;
         rSpare1 : Real;
         rSpare2 : Real;
         rSpare3 : Real;
         rSpare4 : Real;
         rSpare5 : Real;
         rSpare6 : Real;
         rSpare7 : Real;
         rSpare8 : Real;
         tManCmd : Struct
            xJogForward : Bool;   // Carriage manual jog forward {x|x|x|x|O}
            xJogBackward : Bool;   // Carriage manual jog backward {x|x|x|x|O}
            xSpare2 { ExternalWritable := 'False'} : Bool;
            xSpare3 { ExternalWritable := 'False'} : Bool;
            xSpare4 { ExternalWritable := 'False'} : Bool;
            xSpare5 { ExternalWritable := 'False'} : Bool;
            xSpare6 { ExternalWritable := 'False'} : Bool;
            xSpare7 { ExternalWritable := 'False'} : Bool;
            xSpare8 { ExternalWritable := 'False'} : Bool;
            xSpare9 { ExternalWritable := 'False'} : Bool;
            xSpare10 { ExternalWritable := 'False'} : Bool;
            xSpare11 { ExternalWritable := 'False'} : Bool;
            xSpare12 { ExternalWritable := 'False'} : Bool;
            xSpare13 { ExternalWritable := 'False'} : Bool;
            xSpare14 { ExternalWritable := 'False'} : Bool;
            xSpare15 { ExternalWritable := 'False'} : Bool;
            xSpare16 : Bool;
            xSpare17 : Bool;
            xSpare18 : Bool;
            xSpare19 : Bool;
            xSpare20 : Bool;
            xSpare21 : Bool;
            xSpare22 : Bool;
            xSpare23 : Bool;
            xSpare24 : Bool;
            xSpare25 : Bool;
            xSpare26 : Bool;
            xSpare27 : Bool;
            xSpare28 : Bool;
            xSpare29 : Bool;
            xSpare30 : Bool;
            xSpare31 : Bool;
         END_STRUCT;
      END_STRUCT;
   END_STRUCT;


BEGIN

END_DATA_BLOCK

